{attribute 'qualified_only'}
{attribute 'strict'}
TYPE E_MC :
(
	Idle,
	
	RestartCall,
	RestartEffect,
	PowerCall,
	PowerEffect,
	
	HomingCallStep,   
	HomingEffectStep,
	HomingCallServo,   
	HomingEffectServo,
	Execute,
	
	CoupleCallStepMaster,
	CoupleEffectStepMaster,
	MoveAbsCallStepMaster,
	MoveAbsEffectStepMaster,
	DecoupleCallStepMaster,
	DecoupleEffectStepMaster,
	
	
	CoupleCallServoMaster,
	CoupleEffectServoMaster,
	MoveAbsCallServoMaster,
	MoveAbsEffectServoMaster,
	DecoupleCallServoMaster,
	DecoupleEffectServoMaster,
	
	DecoupleCallOnReset,
	DecoupleEffectOnReset,	
	RestartCallOnReset,
	RestartEffectOnReset,	
	
	Error
);
END_TYPE

(* stored: Version 1.1.0.1, ProductVersion 3.1.4024.13
   DUT E_MC: Id {5a8aa116-8988-4c54-9c97-7874ed0f2b92} *)
